FUNCTION BOOLS_TO_DWORD
  (* Standard: 61499-1 *)
  (* Version 1.0, 2024-02-22, franz *)
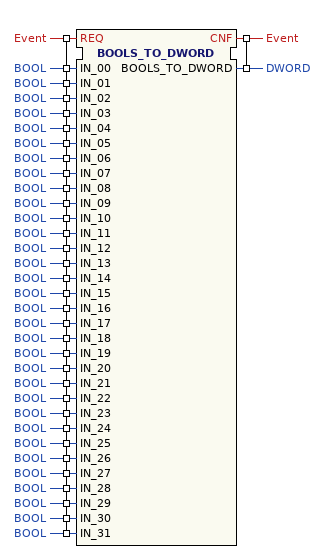
  EVENT_INPUT
    REQ WITH IN_00, IN_01, IN_02, IN_03, IN_04, IN_05, IN_06, IN_07, IN_08, IN_09, IN_10, IN_11, IN_12, IN_13, IN_14, IN_15, IN_16, IN_17, IN_18, IN_19, IN_20, IN_21, IN_22, IN_23, IN_24, IN_25, IN_26, IN_27, IN_28, IN_29, IN_30, IN_31;
  END_EVENT
  EVENT_OUTPUT
    CNF WITH BOOLS_TO_DWORD;
  END_EVENT
  VAR_INPUT
    IN_00 : BOOL; (* BIT 00 *)
    IN_01 : BOOL; (* BIT 01 *)
    IN_02 : BOOL; (* BIT 02 *)
    IN_03 : BOOL; (* BIT 03 *)
    IN_04 : BOOL; (* BIT 04 *)
    IN_05 : BOOL; (* BIT 05 *)
    IN_06 : BOOL; (* BIT 06 *)
    IN_07 : BOOL; (* BIT 07 *)
    IN_08 : BOOL; (* BIT 08 *)
    IN_09 : BOOL; (* BIT 09 *)
    IN_10 : BOOL; (* BIT 10 *)
    IN_11 : BOOL; (* BIT 11 *)
    IN_12 : BOOL; (* BIT 12 *)
    IN_13 : BOOL; (* BIT 13 *)
    IN_14 : BOOL; (* BIT 14 *)
    IN_15 : BOOL; (* BIT 15 *)
    IN_16 : BOOL; (* BIT 16 *)
    IN_17 : BOOL; (* BIT 17 *)
    IN_18 : BOOL; (* BIT 18 *)
    IN_19 : BOOL; (* BIT 19 *)
    IN_20 : BOOL; (* BIT 20 *)
    IN_21 : BOOL; (* BIT 21 *)
    IN_22 : BOOL; (* BIT 22 *)
    IN_23 : BOOL; (* BIT 23 *)
    IN_24 : BOOL; (* BIT 24 *)
    IN_25 : BOOL; (* BIT 25 *)
    IN_26 : BOOL; (* BIT 26 *)
    IN_27 : BOOL; (* BIT 27 *)
    IN_28 : BOOL; (* BIT 28 *)
    IN_29 : BOOL; (* BIT 29 *)
    IN_30 : BOOL; (* BIT 30 *)
    IN_31 : BOOL; (* BIT 31 *)
  END_VAR
  VAR_OUTPUT
    BOOLS_TO_DWORD : DWORD;
  END_VAR
  BODY IN ST:
FUNCTION BOOLS_TO_DWORD : DWORD

VAR_INPUT
	IN_00 : BOOL;    // BIT 00
	IN_01 : BOOL;    // BIT 01
	IN_02 : BOOL;    // BIT 02
	IN_03 : BOOL;    // BIT 03
	IN_04 : BOOL;    // BIT 04
	IN_05 : BOOL;    // BIT 05
	IN_06 : BOOL;    // BIT 06
	IN_07 : BOOL;    // BIT 07
	IN_08 : BOOL;    // BIT 08
	IN_09 : BOOL;    // BIT 09
	IN_10 : BOOL;    // BIT 10
	IN_11 : BOOL;    // BIT 11
	IN_12 : BOOL;    // BIT 12
	IN_13 : BOOL;    // BIT 13
	IN_14 : BOOL;    // BIT 14
	IN_15 : BOOL;    // BIT 15
	IN_16 : BOOL;    // BIT 16
	IN_17 : BOOL;    // BIT 17
	IN_18 : BOOL;    // BIT 18
	IN_19 : BOOL;    // BIT 19
	IN_20 : BOOL;    // BIT 20
	IN_21 : BOOL;    // BIT 21
	IN_22 : BOOL;    // BIT 22
	IN_23 : BOOL;    // BIT 23
	IN_24 : BOOL;    // BIT 24
	IN_25 : BOOL;    // BIT 25
	IN_26 : BOOL;    // BIT 26
	IN_27 : BOOL;    // BIT 27
	IN_28 : BOOL;    // BIT 28
	IN_29 : BOOL;    // BIT 29
	IN_30 : BOOL;    // BIT 30
	IN_31 : BOOL;    // BIT 31
END_VAR

(* this Function combines the 32 BOOLS to a dword *)
BOOLS_TO_DWORD.0 := IN_00;
BOOLS_TO_DWORD.1 := IN_01;
BOOLS_TO_DWORD.2 := IN_02;
BOOLS_TO_DWORD.3 := IN_03;
BOOLS_TO_DWORD.4 := IN_04;
BOOLS_TO_DWORD.5 := IN_05;
BOOLS_TO_DWORD.6 := IN_06;
BOOLS_TO_DWORD.7 := IN_07;
BOOLS_TO_DWORD.8 := IN_08;
BOOLS_TO_DWORD.9 := IN_09;
BOOLS_TO_DWORD.10 := IN_10;
BOOLS_TO_DWORD.11 := IN_11;
BOOLS_TO_DWORD.12 := IN_12;
BOOLS_TO_DWORD.13 := IN_13;
BOOLS_TO_DWORD.14 := IN_14;
BOOLS_TO_DWORD.15 := IN_15;
BOOLS_TO_DWORD.16 := IN_16;
BOOLS_TO_DWORD.17 := IN_17;
BOOLS_TO_DWORD.18 := IN_18;
BOOLS_TO_DWORD.19 := IN_19;
BOOLS_TO_DWORD.20 := IN_20;
BOOLS_TO_DWORD.21 := IN_21;
BOOLS_TO_DWORD.22 := IN_22;
BOOLS_TO_DWORD.23 := IN_23;
BOOLS_TO_DWORD.24 := IN_24;
BOOLS_TO_DWORD.25 := IN_25;
BOOLS_TO_DWORD.26 := IN_26;
BOOLS_TO_DWORD.27 := IN_27;
BOOLS_TO_DWORD.28 := IN_28;
BOOLS_TO_DWORD.29 := IN_29;
BOOLS_TO_DWORD.30 := IN_30;
BOOLS_TO_DWORD.31 := IN_31;
END_FUNCTION
  END_BODY
END_FUNCTION
